KUKA KRL data list: up2.dat

&ACCESS RVP2
&COMMENT Praegen VW310-6
&PARAM DISKPATH = KRC:\R1\UPs
&PARAM TEMPLATE = C:\KRC\Roboter\Template\upvorgabe
&PARAM TPVW_VERSION = 8.1.8
&PARAM EDITMASK = Up999[1-999]
DEFDAT UP2
; FOLD ;%{H} %MKUKATPVW
; ENDFOLD
; interface to basic routines
 EXT  BAS (BAS_COMMAND  :IN,REAL  :IN )
; interface to VW-standard routines
EXT VW (VW_COMMAND:IN, BOOL: IN, REAL:IN, REAL:IN, REAL:IN, REAL:IN, BOOL :IN, E6POS :IN )
; interface to VW_USER - Call
EXT  VW_USER (VW_USER_CMD :IN,INT :IN,REAL  :IN,REAL  :IN,REAL  :IN,REAL  :IN,REAL  :IN,REAL  :IN,BOOL  :IN )
EXT  VW_USR_R (VW_USER_CMD :IN,INT :IN,REAL  :IN,REAL  :IN,REAL  :IN,REAL  :IN,REAL  :IN,REAL  :IN,BOOL  :IN )
EXT  IBGN (IBGN_COMMAND  :IN,BOOL  :IN,REAL  :IN,REAL  :IN,BOOL  :IN,E6POS  :OUT )
; interface select routine
EXTFCT INT  SELECT (SUBTYPE  :IN,INT  :IN,BOOL  :IN,ARI_TYP  :IN,INT  :IN,BOOL_TYP  :IN,INT  :IN,BOOL  :IN)
INT VW_NEXT_FREE = 23
INT VW_NFREE_SPS = 23
INT VW_MAX_SPS = 123
DECL VW_MPARA_TYP P1_D = {TOOL_NO 8,BASE_NO 23,VB 100,VE 0,ACC 100,TRG_TIME 0,MOVE_TYPE #PTP_MOTION}
DECL E6POS P1 = {X 1103.06, Y -1105.41, Z -1619.29, A -89.827, B 60.001, C -104.622, S 2, T 42 , E1 0.0, E2 0.0, E3 0.0, E4 0.0, E5 0.0, E6 0.0}
DECL VW_MPARA_TYP P2_D = {TOOL_NO 8,BASE_NO 23,VB 100,VE 100,ACC 100,TRG_TIME 0,MOVE_TYPE #PTP_MOTION}
DECL E6POS P2 = {X 1772.01, Y -1101.6, Z -718.32, A -76.143, B 5.8, C -48.277, S 2, T 34 , E1 0.0, E2 0.0, E3 0.0, E4 0.0, E5 0.0, E6 0.0}
DECL VW_MPARA_TYP P3_D = {TOOL_NO 8,BASE_NO 23,VB 100,VE 100,ACC 100,TRG_TIME 0,MOVE_TYPE #PTP_MOTION}
DECL E6POS P3 = {X 1054.62, Y 268.14, Z -54.97, A -106.653, B -6.931, C -55.966, S 2, T 42 , E1 0.0, E2 0.0, E3 0.0, E4 0.0, E5 0.0, E6 0.0}
DECL VW_MPARA_TYP P4_D = {TOOL_NO 8,BASE_NO 23,VB 100,VE 100,ACC 100,TRG_TIME 0,MOVE_TYPE #PTP_MOTION}
DECL E6POS P4 = {X 1324.93, Y 627.41, Z 17.73, A -103.707, B -2.88, C -52.636, S 2, T 42 , E1 0.0, E2 0.0, E3 0.0, E4 0.0, E5 0.0, E6 0.0}
DECL VW_MPARA_TYP P5_D = {TOOL_NO 8,BASE_NO 23,VB 100,VE 100,ACC 100,TRG_TIME 0,MOVE_TYPE #PTP_MOTION}
DECL E6POS P5 = {X 1443.17, Y 764.94, Z 359.73, A -97.372, B -3.116, C -68.781, S 2, T 42 , E1 0.0, E2 0.0, E3 0.0, E4 0.0, E5 0.0, E6 0.0}
DECL VW_MPARA_TYP P6_D = {TOOL_NO 8,BASE_NO 23,VB 100,VE 100,ACC 100,TRG_TIME 0,MOVE_TYPE #PTP_MOTION}
DECL E6POS P6 = {X 1647.9, Y 702.7, Z 670.23, A -99.981, B -0.345, C -88.947, S 2, T 42 , E1 0.0, E2 0.0, E3 0.0, E4 0.0, E5 0.0, E6 0.0}
DECL VW_MPARA_TYP P7_D = {TOOL_NO 8,BASE_NO 23,VB 100,VE 100,ACC 100,TRG_TIME 0,MOVE_TYPE #PTP_MOTION}
DECL E6POS P7 = {X 1786.95, Y 695.54, Z 664.93, A -94.981, B -0.436, C -94.981, S 2, T 42 , E1 0.0, E2 0.0, E3 0.0, E4 0.0, E5 0.0, E6 0.0}
DECL VW_MPARA_TYP P8_D = {TOOL_NO 8,BASE_NO 23,VB 100,VE 100,ACC 100,TRG_TIME 0,MOVE_TYPE #PTP_MOTION}
DECL E6POS P8 = {X 1833.94, Y 728.48, Z 645.76, A -90.0, B 0.0, C -95.0, S 2, T 42 , E1 0.0, E2 0.0, E3 0.0, E4 0.0, E5 0.0, E6 0.0}
DECL VW_MPARA_TYP P9_D = {TOOL_NO 8,BASE_NO 23,VB 150,VE 0,ACC 100,TRG_TIME 5,MOVE_TYPE #PATH_MOTION}
DECL E6POS P9 = {X 1833.95, Y 741.47, Z 645.74, A -90.0, B 0.001, C -95.0, S 2, T 42 , E1 0.0, E2 0.0, E3 0.0, E4 0.0, E5 0.0, E6 0.0}
DECL VW_MPARA_TYP P10_D = {TOOL_NO 8,BASE_NO 23,VB 150,VE 0,ACC 100,TRG_TIME 0,MOVE_TYPE #PATH_MOTION}
DECL E6POS P10 = {X 1833.94, Y 728.48, Z 645.76, A -90.0, B 0.0, C -95.0, S 2, T 42 , E1 0.0, E2 0.0, E3 0.0, E4 0.0, E5 0.0, E6 0.0}
DECL VW_MPARA_TYP P11_D = {TOOL_NO 8,BASE_NO 23,VB 100,VE 100,ACC 100,TRG_TIME 0,MOVE_TYPE #PTP_MOTION}
DECL E6POS P11 = {X 1755.09, Y 705.48, Z 698.66, A -90.0, B 0.0, C -94.982, S 2, T 42 , E1 0.0, E2 0.0, E3 0.0, E4 0.0, E5 0.0, E6 0.0}
DECL VW_MPARA_TYP P12_D = {TOOL_NO 8,BASE_NO 23,VB 100,VE 100,ACC 100,TRG_TIME 0,MOVE_TYPE #PTP_MOTION}
DECL E6POS P12 = {X 1676.06, Y 728.7, Z 421.21, A -90.0, B 0.0, C -69.018, S 2, T 42 , E1 0.0, E2 0.0, E3 0.0, E4 0.0, E5 0.0, E6 0.0}
DECL VW_MPARA_TYP P13_D = {TOOL_NO 8,BASE_NO 23,VB 150,VE 0,ACC 100,TRG_TIME 5,MOVE_TYPE #PATH_MOTION}
DECL E6POS P13 = {X 1676.0, Y 741.7, Z 420.99, A -90.0, B 0.0, C -69.0, S 2, T 42 , E1 0.0, E2 0.0, E3 0.0, E4 0.0, E5 0.0, E6 0.0}
DECL VW_MPARA_TYP P14_D = {TOOL_NO 8,BASE_NO 23,VB 150,VE 0,ACC 100,TRG_TIME 0,MOVE_TYPE #PATH_MOTION}
DECL E6POS P14 = {X 1676.06, Y 728.7, Z 421.21, A -90.0, B 0.0, C -69.018, S 2, T 42 , E1 0.0, E2 0.0, E3 0.0, E4 0.0, E5 0.0, E6 0.0}
DECL VW_MPARA_TYP P15_D = {TOOL_NO 8,BASE_NO 23,VB 100,VE 100,ACC 100,TRG_TIME 0,MOVE_TYPE #PTP_MOTION}
DECL E6POS P15 = {X 1755.09, Y 705.48, Z 698.66, A -90.0, B 0.0, C -94.982, S 2, T 42 , E1 0.0, E2 0.0, E3 0.0, E4 0.0, E5 0.0, E6 0.0}
DECL VW_MPARA_TYP P16_D = {TOOL_NO 8,BASE_NO 23,VB 100,VE 100,ACC 100,TRG_TIME 0,MOVE_TYPE #PTP_MOTION}
DECL E6POS P16 = {X 1786.95, Y 695.54, Z 664.93, A -94.981, B -0.436, C -94.981, S 2, T 42 , E1 0.0, E2 0.0, E3 0.0, E4 0.0, E5 0.0, E6 0.0}
DECL VW_MPARA_TYP P17_D = {TOOL_NO 8,BASE_NO 23,VB 100,VE 100,ACC 100,TRG_TIME 0,MOVE_TYPE #PTP_MOTION}
DECL E6POS P17 = {X 1647.9, Y 702.7, Z 670.23, A -99.981, B -0.345, C -88.947, S 2, T 42 , E1 0.0, E2 0.0, E3 0.0, E4 0.0, E5 0.0, E6 0.0}
DECL VW_MPARA_TYP P18_D = {TOOL_NO 8,BASE_NO 23,VB 100,VE 100,ACC 100,TRG_TIME 0,MOVE_TYPE #PTP_MOTION}
DECL E6POS P18 = {X 1443.17, Y 764.94, Z 359.73, A -97.372, B -3.116, C -68.781, S 2, T 42 , E1 0.0, E2 0.0, E3 0.0, E4 0.0, E5 0.0, E6 0.0}
DECL VW_MPARA_TYP P19_D = {TOOL_NO 8,BASE_NO 23,VB 100,VE 100,ACC 100,TRG_TIME 0,MOVE_TYPE #PTP_MOTION}
DECL E6POS P19 = {X 1324.93, Y 627.41, Z 17.73, A -103.707, B -2.88, C -52.636, S 2, T 42 , E1 0.0, E2 0.0, E3 0.0, E4 0.0, E5 0.0, E6 0.0}
DECL VW_MPARA_TYP P20_D = {TOOL_NO 8,BASE_NO 23,VB 100,VE 100,ACC 100,TRG_TIME 0,MOVE_TYPE #PTP_MOTION}
DECL E6POS P20 = {X 1054.62, Y 268.14, Z -54.97, A -106.653, B -6.931, C -55.966, S 2, T 42 , E1 0.0, E2 0.0, E3 0.0, E4 0.0, E5 0.0, E6 0.0}
DECL VW_MPARA_TYP P21_D = {TOOL_NO 8,BASE_NO 23,VB 100,VE 100,ACC 100,TRG_TIME 0,MOVE_TYPE #PTP_MOTION}
DECL E6POS P21 = {X 1772.0, Y -1101.6, Z -728.32, A -76.143, B 5.8, C -48.277, S 2, T 34 , E1 0.0, E2 0.0, E3 0.0, E4 0.0, E5 0.0, E6 0.0}
DECL VW_MPARA_TYP P22_D = {TOOL_NO 8,BASE_NO 23,VB 100,VE 0,ACC 100,TRG_TIME 0,MOVE_TYPE #PTP_MOTION}
DECL E6POS P22 = {X 1103.06, Y -1105.41, Z -1619.28, A -89.827, B 60.001, C -104.622, S 2, T 42 , E1 0.0, E2 0.0, E3 0.0, E4 0.0, E5 0.0, E6 0.0}
ENDDAT
